(* IEC 61131-3 sources: Caravan/Archiv/12-04-19/Stations/MachineControl/MachineControl/Class/HmiImage35, 1 file *)

(* ---- HmiImage35.st ---- *)
(*!
<Class
	Name               = "HmiImage35"
	Revision           = "0.3"
	RealtimeTask       = "false"
	CyclicTask         = "false"
	BackgroundTask     = "false"
	Sigmatek           = "true"
	OSInterface        = "false"
	HighPriority       = "false"
	Automatic          = "false"
	UpdateMode         = "Prescan"
	SharedCommandTable = "true"
	Objectsize         = "(284,120)">
	<Channels>
		<Server Name="ByteSize" Visualized="false" Initialize="false" WriteProtected="true" Retentive="false"/>
		<Server Name="ClassSvr" Visualized="false" Initialize="false" WriteProtected="true" Retentive="false"/>
		<Client Name="StdLib" Required="false" Internal="false"/>
	</Channels>
	<RevDoku>
		<Owner Company="sigmatek" Author="kolott"/>
		<Dokumentation Revision="0.3" Date="2015-03-04" Author="kolott" Company="sigmatek" Description="name of datatype has changed (_BOX_IMAGELIST --&gt; _BOX_IMAGE) because named is a single image and not a list of images. "/>
		<Dokumentation Revision="0.2" Date="2014-03-26" Author="kolott" Company="sigmatek" Description="innovation: ClassSvr will represent number of generated images for hmi&#13;&#10;server ByteSize added"/>
	</RevDoku>
</Class>
*)
HmiImage35 : CLASS
  //Servers:
	ClassSvr 	: SvrChCmd_DINT;
	ByteSize 	: SvrCh_UDINT;
  //Clients:
	StdLib 	: CltChCmd__StdLib;
  //Variables:
  //Functions:

	FUNCTION GLOBAL CreateList
		VAR_INPUT
			width 	: UDINT;
			height 	: UDINT;
			transparent 	: UINT;
			state 	: UINT;
			datano 	: UDINT;
			dataptr 	: ^void;
		END_VAR
		VAR_OUTPUT
			retcode 	: ^void;
		END_VAR;

	FUNCTION GLOBAL Start;
  //Tables:
	FUNCTION @STD
		VAR_OUTPUT
			ret_code	: CONFSTATES;
		END_VAR;
	FUNCTION GLOBAL TAB @CT_;
END_CLASS;

#pragma usingLtd _StdLib

#includeC "..\LseEasy\Create.h"

#define BMP_NO_COMPRESSION 0x8000

FUNCTION GLOBAL HmiImage35::Start

  ClassSvr := 0;
  ByteSize := 0;

END_FUNCTION

FUNCTION GLOBAL HmiImage35::CreateList
	VAR_INPUT
    width : udint;
    height : udint;
    transparent : uint;
    state : uint;
    datano : udint;
    dataptr : ^void;
	END_VAR
	VAR_OUTPUT
		retcode 	: ^void;
	END_VAR
  VAR
    pbox : ^_BOX_IMAGE;
    size, maxi : udint;
    ph : ^uint;
    xx : uint;
    ppixdat : ^_BMPDAT;
  END_VAR

  retcode := NIL;
  if((datano > 0) & (dataptr <> NIL)) then
    size := datano * 3;
    maxi := width * height * 2;

    if(size < maxi) then
      // image mit lauflängenkomprimierung
      retcode := StdLib.MallocV1(size + sizeof(_BOX_IMAGE) - 1, 0);
      if(retcode <> NIL) then
        pbox$^void              := retcode;
        setup_BIGBOX_HEADER(#pbox^.boxhdr, 0);
        pbox^.image.mp          := 16#504D;
        pbox^.image.datano      := datano;
        pbox^.image.width       := width$uint;
        pbox^.image.height      := height$uint;
        pbox^.image.state       := (state and 16#7FFF);
        pbox^.image.transparent := transparent;
        _memcpy(#pbox^.image.data[0], dataptr, size);
        end_BIGBOX_HEADER(#pbox^.boxhdr, size + sizeof(_BOX_IMAGE) - 1);
      end_if;
    else
      // image ohne lauflängenkomprimierung
      retcode := StdLib.MallocV1(maxi + sizeof(_BOX_IMAGE) - 1, 0);
      if(retcode <> NIL) then
        pbox$^void              := retcode;
        setup_BIGBOX_HEADER(#pbox^.boxhdr, 0);
        pbox^.image.mp          := 16#504D;
        pbox^.image.datano      := width * height;
        pbox^.image.width       := width$uint;
        pbox^.image.height      := height$uint;
        pbox^.image.state       := state or 16#8000; // kennung für lauflängenkomprimierung
        pbox^.image.transparent := transparent;

        ph$^usint     := #pbox^.image.data[0];
        ppixdat$^void := dataptr;
        while(datano) do
          xx := ppixdat^.no;
          while(xx) do
            ph^ := ppixdat^.col;
            xx -= 1;
            ph += 2;
          end_while;
          ppixdat += sizeof(_BMPDAT);
          datano  -= 1;
        end_while;

        end_BIGBOX_HEADER(#pbox^.boxhdr, maxi + sizeof(_BOX_IMAGE) - 1);
      end_if;
    end_if;
  end_if;

  if(retcode <> nil) then
    ClassSvr   += 1;
    pbox$^void := retcode;
    ByteSize   += pbox^.boxhdr.size;
  end_if;

END_FUNCTION
